(* CoDeSys 2.3.9.62 project: Tema1 Ejercicio1.pro *)
(* Libraries: Standard.lib 4.10.05 10:14:46 *)

(* Global variable list: Global_Variables *)
VAR_GLOBAL
(* Entradas *)
      Nivel:BOOL;
      Temp: BOOL;
       Pres:BOOL;
      ACK:BOOL;

(*Salidas*)
      Alarma: BOOL;
       LuzPres:BOOL;
      LuzTemp:BOOL;
      LuzNiv:BOOL;

END_VAR

(* POU PLC_PRG, LD *)
PROGRAM PLC_PRG
VAR

END_VAR
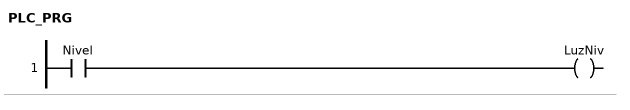
_LD_ (* Ladder Diagram *)
NETWORK 1
	[Nivel] --- (LuzNiv)
_END_LD_
(* the same logic as Structured Text *)
(* Network 1 *)
LuzNiv := Nivel;
END_PROGRAM

(* Visualisation PresNivTemp
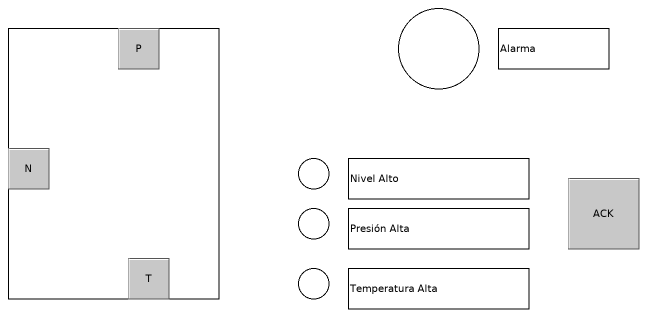
button at (220,310)-(261,351): text "T"; toggles Temp
button at (210,80)-(251,121): text "P"; toggles Pres
button at (100,200)-(141,241): text "N"; toggles Nivel
ellipse at (490,60)-(571,141): alarm colour if Alarma
ellipse at (390,210)-(421,241): alarm colour if LuzNiv
rectangle at (440,210)-(621,251): text "Nivel Alto"
ellipse at (390,260)-(421,291): alarm colour if LuzPres
rectangle at (440,260)-(621,301): text "Presión Alta"
ellipse at (390,320)-(421,351): alarm colour if LuzTemp
rectangle at (440,320)-(621,361): text "Temperatura Alta"
rectangle at (590,80)-(701,121): text "Alarma"
button at (660,230)-(731,301): text "ACK"; taps ACK
1 more shapes without text or variables
*)
